// §3.8e test source: an owner on this controller, with a failure the test can
// switch on. A test seam, so it lives here and never in the library (lint C8).
FUNCTION_BLOCK FB_ProbeLineSource IMPLEMENTS I_LineSource
VAR
    {attribute 'OPC.UA.DA' := '0'}
    _owner : POINTER TO FB_LineData;
    _fail  : BOOL;
END_VAR

;

METHOD Setup : BOOL
VAR_INPUT
    pOwner : POINTER TO FB_LineData;
END_VAR
_owner := pOwner;
Setup := (pOwner <> 0);
END_METHOD

METHOD M_SetFail
VAR_INPUT
    Fail : BOOL;
END_VAR
_fail := Fail;
END_METHOD

METHOD M_Poll : BOOL
VAR_IN_OUT
    Image : ST_LineImage;
END_VAR
M_Poll := FALSE;
IF _fail OR (_owner = 0) THEN
    RETURN;
END_IF
Image := _owner^.Image;
M_Poll := TRUE;
END_METHOD

METHOD M_Error : DINT
M_Error := SEL(_fail, 0, 99);
END_METHOD

END_FUNCTION_BLOCK

(* stored: Version 1.1.0.1, ProductVersion 3.1.4024.12
   POU FB_ProbeLineSource: Id {dc2ca3c6-4eb8-47b0-96c9-67bac286fb7b}, SpecialFunc None
   Method Setup: Id {8e801e45-5c82-4c19-96d0-0e3bc0006205}
   Method M_SetFail: Id {a0c9f82f-7b69-4a5d-af86-6a3aa74e4665}
   Method M_Poll: Id {3fb50aee-115b-4781-b14f-6756e2bf1a9e}
   Method M_Error: Id {253e4237-27a7-4f65-a982-95ed05437833} *)
